# EPICS substitutions: CsHeaterApp/Db/Watlow_PM_IOC_Alarm.substitutions
file Watlow_PM_IOC_Alarm.template
{
pattern	{  s, ta,      ss}
	{   , SE,  Watlow}
}

file save_restoreStatus.db
{
pattern {P}
        {:CS:Watlow:}
}

file ioc_sns.db
{
pattern {IOCNAME}
        {:CS:Watlow}
}
